PROGRAM EStop
VAR			
	estop_oneleft: ARRAY [1..5] OF WORD := [16#2A2A, 16#2A45, 16#4D45, 16#5247, 16#454E];
	estop_oneright: ARRAY [1..5] OF WORD := [16#4359, 16#2053, 16#544F, 16#502A, 16#2A2A];
	
	remote: ARRAY [1..5] OF WORD := [16#5265, 16#6D6F, 16#7465, 16#2020, 16#2020];
	pit: ARRAY [1..5] OF WORD := [16#5069, 16#7420, 16#2020, 16#2020, 16#2020];
	pump: ARRAY [1..5] OF WORD := [16#5075, 16#6D70, 16#2020, 16#2020, 16#2020];
	upstage: ARRAY [1..5] OF WORD := [16#5570, 16#7374, 16#6167, 16#6520, 16#2020];
	downstage: ARRAY [1..5] OF WORD := [16#446F, 16#776E, 16#7374, 16#6167, 16#6520];
	console: ARRAY [1..5] OF WORD := [16#436F, 16#6E73, 16#6F6C, 16#6520, 16#2020];
	
	pageNum: WORD := 0;	
END_VAR

IF GV_MODBUS.btnData = GV_MODBUS.btnUp THEN
	pageNum := 0;
	Execute_Write_Screen();
END_IF

IF GV_MODBUS.btnData = GV_MODBUS.btnDwn THEN
	pageNum := 1;
	Execute_Write_Screen();
END_IF

IF pageNum = 0 THEN
	GV_MODBUS.oneLeft:= estop_oneleft;
	GV_MODBUS.oneRight:= estop_oneright;   
                           
	GV_MODBUS.twoLeft:= remote;
	IF GV_LIFT.REMOTE_ESTOP_INDICATOR_OUT THEN
		GV_MODBUS.twoRight:= GV_MODBUS.engaged;
	ELSE
		GV_MODBUS.twoRight:= GV_MODBUS.ok;
	END_IF  
                            
	GV_MODBUS.threeLeft:= pit;
	IF GV_LIFT.PIT_ESTOP_INDICATOR_OUT THEN
		GV_MODBUS.threeRight:= GV_MODBUS.engaged;
	ELSE
		GV_MODBUS.threeRight:= GV_MODBUS.ok;
	END_IF	
                               
	GV_MODBUS.fourLeft:= pump; 
	IF GV_LIFT.PUMP_ESTOP_INDICATOR_OUT THEN
		GV_MODBUS.fourRight:= GV_MODBUS.engaged;
	ELSE
		GV_MODBUS.fourRight:= GV_MODBUS.ok;		
	END_IF
END_IF

IF pageNum = 1 THEN
	GV_MODBUS.oneLeft:= estop_oneleft;
	GV_MODBUS.oneRight:= estop_oneright;   
                           
	GV_MODBUS.twoLeft:= downstage;
	IF GV_LIFT.DOWNSTAGE_ESTOP_INDICATOR_OUT THEN
		GV_MODBUS.twoRight:= GV_MODBUS.engaged;
	ELSE
		GV_MODBUS.twoRight:= GV_MODBUS.ok;
	END_IF
                            
	GV_MODBUS.threeLeft:= upstage;
	IF GV_LIFT.UPSTAGE_ESTOP_INDICATOR_OUT THEN
		GV_MODBUS.threeRight:= GV_MODBUS.engaged;
	ELSE
		GV_MODBUS.threeRight:= GV_MODBUS.ok;
	END_IF
                               
	GV_MODBUS.fourLeft:= console; 
	IF GV_LIFT.CONSOLE_ESTOP_INDICATOR_OUT THEN
		GV_MODBUS.fourRight:= GV_MODBUS.engaged;
	ELSE
		GV_MODBUS.fourRight:= GV_MODBUS.ok;
	END_IF
END_IF

IF NOT GV_MODBUS.readExecute AND GV_MODBUS.addr = GV_MODBUS.oneLeftAddr THEN
	GV_MODBUS.data:= GV_MODBUS.oneLeft;
END_IF

END_PROGRAM

(* stored: Version 1.1.0.1, ProductVersion 3.1.4022.12
   POU EStop: Id {7a8665f7-e86e-4807-86a9-336a6c1b3fd4}, SpecialFunc None *)
